# B&R Automation Studio project MotionTestBenchMaster (part 56)

```iecst
                               VAR_DOS_SEQ.Device.LTJ203.ALR_HighLimitEn := FALSE;                                     (* STEP: 115 Hema Tank Level*)
                               VAR_DOS_SEQ.Device.LTJ203.ALR_HighLimitSP := 0;
                               VAR_DOS_SEQ.Device.LTJ203.ALR_LowLimitEn := FALSE;
                               VAR_DOS_SEQ.Device.LTJ203.ALR_LowLimitSP := 0;
                               VAR_DOS_SEQ.Device.LTJ203.SP := 0;
                               VAR_DOS_SEQ.Device.LTJ203.CMP := 0;
                               VAR_DOS_SEQ.Device.LTJ203.MinDev := 0;
                               VAR_DOS_SEQ.Device.LTJ203.MaxDev := 0;

                               VAR_DOS_SEQ.Device.TTJ203.ALR_HighLimitEn := FALSE;                                     (* STEP: 115 Hema Tank Temperature*)
                               VAR_DOS_SEQ.Device.TTJ203.ALR_HighLimitSP := 0;
                               VAR_DOS_SEQ.Device.TTJ203.ALR_LowLimitEn := FALSE;
                               VAR_DOS_SEQ.Device.TTJ203.ALR_LowLimitSP := 0;
                               VAR_DOS_SEQ.Device.TTJ203.SP := 0;
                               VAR_DOS_SEQ.Device.TTJ203.CMP := 0;
                               VAR_DOS_SEQ.Device.TTJ203.MinDev := 0;
                               VAR_DOS_SEQ.Device.TTJ203.MaxDev := 0;

                               VAR_DOS_SEQ.Device.LSJ200.ALR := FALSE;                                                 (* STEP: 115 *)
                               VAR_DOS_SEQ.Device.LSJ200.WAIT_OFF := FALSE;
                               VAR_DOS_SEQ.Device.LSJ200.WAIT_ON := FALSE;

                               VAR_DOS_SEQ.Device.LSJ201.ALR := FALSE;                                                 (* STEP: 115 *)
                               VAR_DOS_SEQ.Device.LSJ201.WAIT_OFF := FALSE;
                               VAR_DOS_SEQ.Device.LSJ201.WAIT_ON := FALSE;

                               VAR_DOS_SEQ.Device.LSJ202.ALR := FALSE;                                                 (* STEP: 115 *)
                               VAR_DOS_SEQ.Device.LSJ202.WAIT_OFF := FALSE;
                               VAR_DOS_SEQ.Device.LSJ202.WAIT_ON := FALSE;

                               VAR_DOS_SEQ.Device.FSJ201.ALR := FALSE;                                                 (* STEP: 115 *)
                               VAR_DOS_SEQ.Device.FSJ201.WAIT_OFF := FALSE;
                               VAR_DOS_SEQ.Device.FSJ201.WAIT_ON := FALSE;

                               VAR_DOS_SEQ.Device.FSJ202.ALR := FALSE;                                                 (* STEP: 115 *)
                               VAR_DOS_SEQ.Device.FSJ202.WAIT_OFF := FALSE;
                               VAR_DOS_SEQ.Device.FSJ202.WAIT_ON := FALSE;

                               VAR_DOS_SEQ.Mem.PBAbortEnable := TRUE;                                                  (* STEP: 115 PB Abort Sequence Enable*)
                               VAR_DOS_SEQ.Mem.PBStopEnable := FALSE;                                                  (* STEP: 115 PB Stop Sequence Enable*)
                               VAR_DOS_SEQ.Mem.PBStartEnable := FALSE;                                                 (* STEP: 115 PB Start Sequence Enable*)
                               VAR_DOS_SEQ.Mem.ContainersStop := TRUE;                                                 (* STEP: 115 *)
                               VAR_DOS_SEQ.Mem.MachineStart := FALSE;                                                  (* STEP: 115 *)
                               VAR_DOS_SEQ.Mem.MachineStop := TRUE;                                                    (* STEP: 115 *)
                               VAR_DOS_SEQ.Mem.DummyBottles := FALSE;                                                  (* STEP: 115 Dummy Bottle Install*)
                               VAR_DOS_SEQ.Mem.PositioningRequest := FALSE;                                            (* STEP: 115 Request of Cam Positioning at height SP of Sequncer*)
                               VAR_DOS_SEQ.Mem.COP_Cycle := FALSE;                                                     (* STEP: 115 COP Cycle Check Requested*)
                               VAR_DOS_SEQ.Mem.LapsCounter := FALSE;                                                   (* STEP: 115 *)
                               VAR_DOS_SEQ.Mem.ValveOpening := FALSE;                                                  (* STEP: 115 *)
                               VAR_DOS_SEQ.Mem.CopAfterCipRequest := FALSE;                                            (* STEP: 115 Request Of Cop After Cip*)

                               VAR_DOS_SEQ.ITC.CIP_CleaningRequest := FALSE;                                           (* STEP: 115 To CIP -> Request of Solution Sending*)
                               VAR_DOS_SEQ.ITC.CIP_Alarm := FALSE;                                                     (* STEP: 115 To CIP -> Critical Alarm Present*)
                               VAR_DOS_SEQ.ITC.CIP_RinseEnded := FALSE;                                                (* STEP: 115 To CIP -> Rinse Finished*)
                               VAR_DOS_SEQ.ITC.CIP_ChangeEnded := FALSE;                                               (* STEP: 115 To CIP -> Change Finished*)
                               VAR_DOS_SEQ.ITC.CIP_DrainRunning := FALSE;                                              (* STEP: 115 To CIP -> Drain Cycle Running*)
                               VAR_DOS_SEQ.ITC.CIP_RinseRunning := FALSE;                                              (* STEP: 115 To CIP -> Rinse Cycle Running*)
                               VAR_DOS_SEQ.ITC.CIP_CleaningRunning := FALSE;                                           (* STEP: 115 To CIP -> Cleaning Cycle Running*)
                               VAR_DOS_SEQ.ITC.CIP_DrainEnded := FALSE;                                                (* STEP: 115 To CIP -> Drain Finished*)
                               VAR_DOS_SEQ.ITC.CIP_FloodingEnded := FALSE;                                             (* STEP: 115 To CIP -> Flooding Finished*)
                               VAR_DOS_SEQ.ITC.CIP_FlipEnable := FALSE;                                                (* STEP: 115 *)
                               VAR_DOS_SEQ.ITC.CIP_CycleEnded := FALSE;                                                (* STEP: 115 *)

                               VAR_DOS_SEQ.ITC.PROD_ReadyForHeating := FALSE;                                          (* STEP: 115 To PASTO -> Filler Ready for Production (Heating)*)
                               VAR_DOS_SEQ.ITC.PROD_DoserInTemperature := FALSE;                                       (* STEP: 115 To PASTO -> Filler Temperature OK (After Heating)*)
                               VAR_DOS_SEQ.ITC.PROD_ProductRequest := FALSE;                                           (* STEP: 115 To PASTO -> Product Request*)
                               VAR_DOS_SEQ.ITC.PROD_DoserOnFillingMode := FALSE;                                       (* STEP: 115 To PASTO -> Product Consumend -Filling Valve Opening*)
                               VAR_DOS_SEQ.ITC.PROD_EndProductionCompleted := FALSE;                                   (* STEP: 115 To PASTO -> End Production Done*)
                               VAR_DOS_SEQ.ITC.PROD_ProductRecoveryEnd := FALSE;                                       (* STEP: 115 To PASTO -> Product Recovery End*)
                               VAR_DOS_SEQ.ITC.PROD_WaterRequestAfterProd := FALSE;                                    (* STEP: 115 To PASTO -> Water Request For Filler Rinse Afetr Production*)

                       116..129: (* Spare Steps *)

                       130: (* DRAIN - Final Drain *)

                               VAR_DOS_SEQ.Device.PPJ201_PID.PID_Enable := FALSE;                                      (* STEP: 130 Doser Recovery Pump*)
                               VAR_DOS_SEQ.Device.PPJ201_PID.PID_Mode := FALSE;
                               VAR_DOS_SEQ.Device.PPJ201_PID.Auto_SP_Value := 0;
                               VAR_DOS_SEQ.Device.PPJ201_PID.FIX_Value := 0;

                               VAR_DOS_SEQ.Device.PPJ202_PID.PID_Enable := FALSE;                                      (* STEP: 130 Doser Recovery Pump*)
                               VAR_DOS_SEQ.Device.PPJ202_PID.PID_Mode := FALSE;
                               VAR_DOS_SEQ.Device.PPJ202_PID.Auto_SP_Value := 0;
                               VAR_DOS_SEQ.Device.PPJ202_PID.FIX_Value := 0;

                               VAR_DOS_SEQ.Device.PPJ203_PID.PID_Enable := FALSE;                                      (* STEP: 130 Diaphragm Pump for Recovery pulp*)
                               VAR_DOS_SEQ.Device.PPJ203_PID.PID_Mode := FALSE;
                               VAR_DOS_SEQ.Device.PPJ203_PID.Auto_SP_Value := 0;
                               VAR_DOS_SEQ.Device.PPJ203_PID.FIX_Value := 0;

                               VAR_DOS_SEQ.Device.MMJ201_PID.PID_Enable := FALSE;                                      (* STEP: 130 Shaker Motor*)
                               VAR_DOS_SEQ.Device.MMJ201_PID.PID_Mode := FALSE;
                               VAR_DOS_SEQ.Device.MMJ201_PID.Auto_SP_Value := 0;
                               VAR_DOS_SEQ.Device.MMJ201_PID.FIX_Value := 0;

                               VAR_DOS_SEQ.Device.RVJ201_PID.PID_Enable := FALSE;                                      (* STEP: 130 *)
                               VAR_DOS_SEQ.Device.RVJ201_PID.PID_Mode := FALSE;
                               VAR_DOS_SEQ.Device.RVJ201_PID.Auto_SP_Value := 0;
                               VAR_DOS_SEQ.Device.RVJ201_PID.FIX_Value := 0;

                               VAR_DOS_SEQ.Device.AVJ201.AutoCnd := FALSE;                                             (* STEP: 130 Inlet Valve*)
                               VAR_DOS_SEQ.Device.AVJ201.EnableCnd := FALSE;
                               VAR_DOS_SEQ.Device.AVJ210.AutoCnd := FALSE;                                             (* STEP: 130 Washing Duct Valve*)
                               VAR_DOS_SEQ.Device.AVJ210.EnableCnd := FALSE;
                               VAR_DOS_SEQ.Device.AVJ211.AutoCnd := FALSE;                                             (* STEP: 130 Sprayball Valve*)
                               VAR_DOS_SEQ.Device.AVJ211.EnableCnd := FALSE;
                               VAR_DOS_SEQ.Device.AVJ212.AutoCnd := FALSE;                                             (* STEP: 130 *)
                               VAR_DOS_SEQ.Device.AVJ212.EnableCnd := FALSE;
                               VAR_DOS_SEQ.Device.AVJ215.AutoCnd := TRUE;                                              (* STEP: 130 Atmospheric drain valve*)
                               VAR_DOS_SEQ.Device.AVJ215.EnableCnd := FALSE;
                               VAR_DOS_SEQ.Device.AVJ216.AutoCnd := FALSE;                                             (* STEP: 130 Recirculation Valve*)
                               VAR_DOS_SEQ.Device.AVJ216.EnableCnd := FALSE;
                               VAR_DOS_SEQ.Device.AVJ217.AutoCnd := TRUE;                                              (* STEP: 130 Tank Hema Drain Valve*)
                               VAR_DOS_SEQ.Device.AVJ217.EnableCnd := FALSE;
                               VAR_DOS_SEQ.Device.AVJ218.AutoCnd := FALSE;                                             (* STEP: 130 Recirculation Valve*)
                               VAR_DOS_SEQ.Device.AVJ218.EnableCnd := FALSE;
                               VAR_DOS_SEQ.Device.AVJ221.AutoCnd := TRUE;                                              (* STEP: 130 Inlet Loop Valve*)
                               VAR_DOS_SEQ.Device.AVJ221.EnableCnd := FALSE;
                               VAR_DOS_SEQ.Device.AVJ230.AutoCnd := FALSE;                                             (* STEP: 130 *)
                               VAR_DOS_SEQ.Device.AVJ230.EnableCnd := FALSE;
                               VAR_DOS_SEQ.Device.AVJ231.AutoCnd := FALSE;                                             (* STEP: 130 *)
                               VAR_DOS_SEQ.Device.AVJ231.EnableCnd := FALSE;
                               VAR_DOS_SEQ.Device.AVJ232.AutoCnd := TRUE;                                              (* STEP: 130 *)
                               VAR_DOS_SEQ.Device.AVJ232.EnableCnd := FALSE;
                               VAR_DOS_SEQ.Device.AVJ233.AutoCnd := FALSE;                                             (* STEP: 130 *)
                               VAR_DOS_SEQ.Device.AVJ233.EnableCnd := FALSE;
                               VAR_DOS_SEQ.Device.AVJ234.AutoCnd := FALSE;                                             (* STEP: 130 *)
                               VAR_DOS_SEQ.Device.AVJ234.EnableCnd := FALSE;
                               VAR_DOS_SEQ.Device.AVJ235.AutoCnd := FALSE;                                             (* STEP: 130 *)
                               VAR_DOS_SEQ.Device.AVJ235.EnableCnd := FALSE;

                               VAR_DOS_SEQ.Device.LTJ203.ALR_HighLimitEn := FALSE;                                     (* STEP: 130 Hema Tank Level*)
                               VAR_DOS_SEQ.Device.LTJ203.ALR_HighLimitSP := 0;
                               VAR_DOS_SEQ.Device.LTJ203.ALR_LowLimitEn := FALSE;
                               VAR_DOS_SEQ.Device.LTJ203.ALR_LowLimitSP := 0;
                               VAR_DOS_SEQ.Device.LTJ203.SP := 0;
                               VAR_DOS_SEQ.Device.LTJ203.CMP := 0;
                               VAR_DOS_SEQ.Device.LTJ203.MinDev := 0;
                               VAR_DOS_SEQ.Device.LTJ203.MaxDev := 0;

                               VAR_DOS_SEQ.Device.TTJ203.ALR_HighLimitEn := FALSE;                                     (* STEP: 130 Hema Tank Temperature*)
                               VAR_DOS_SEQ.Device.TTJ203.ALR_HighLimitSP := 0;
                               VAR_DOS_SEQ.Device.TTJ203.ALR_LowLimitEn := FALSE;
                               VAR_DOS_SEQ.Device.TTJ203.ALR_LowLimitSP := 0;
                               VAR_DOS_SEQ.Device.TTJ203.SP := 0;
                               VAR_DOS_SEQ.Device.TTJ203.CMP := 0;
                               VAR_DOS_SEQ.Device.TTJ203.MinDev := 0;
                               VAR_DOS_SEQ.Device.TTJ203.MaxDev := 0;

                               VAR_DOS_SEQ.Device.LSJ200.ALR := FALSE;                                                 (* STEP: 130 *)
                               VAR_DOS_SEQ.Device.LSJ200.WAIT_OFF := FALSE;
                               VAR_DOS_SEQ.Device.LSJ200.WAIT_ON := FALSE;

                               VAR_DOS_SEQ.Device.LSJ201.ALR := FALSE;                                                 (* STEP: 130 *)
                               VAR_DOS_SEQ.Device.LSJ201.WAIT_OFF := FALSE;
                               VAR_DOS_SEQ.Device.LSJ201.WAIT_ON := FALSE;

                               VAR_DOS_SEQ.Device.LSJ202.ALR := FALSE;                                                 (* STEP: 130 *)
                               VAR_DOS_SEQ.Device.LSJ202.WAIT_OFF := FALSE;
                               VAR_DOS_SEQ.Device.LSJ202.WAIT_ON := FALSE;

                               VAR_DOS_SEQ.Device.FSJ201.ALR := FALSE;                                                 (* STEP: 130 *)
                               VAR_DOS_SEQ.Device.FSJ201.WAIT_OFF := FALSE;
                               VAR_DOS_SEQ.Device.FSJ201.WAIT_ON := FALSE;

                               VAR_DOS_SEQ.Device.FSJ202.ALR := FALSE;                                                 (* STEP: 130 *)
                               VAR_DOS_SEQ.Device.FSJ202.WAIT_OFF := FALSE;
                               VAR_DOS_SEQ.Device.FSJ202.WAIT_ON := FALSE;

                               VAR_DOS_SEQ.Mem.PBAbortEnable := TRUE;                                                  (* STEP: 130 PB Abort Sequence Enable*)
                               VAR_DOS_SEQ.Mem.PBStopEnable := TRUE;                                                   (* STEP: 130 PB Stop Sequence Enable*)
                               VAR_DOS_SEQ.Mem.PBStartEnable := FALSE;                                                 (* STEP: 130 PB Start Sequence Enable*)
                               VAR_DOS_SEQ.Mem.ContainersStop := TRUE;                                                 (* STEP: 130 *)
                               VAR_DOS_SEQ.Mem.MachineStart := TRUE;                                                   (* STEP: 130 *)
                               VAR_DOS_SEQ.Mem.MachineStop := FALSE;                                                   (* STEP: 130 *)
                               VAR_DOS_SEQ.Mem.DummyBottles := FALSE;                                                  (* STEP: 130 Dummy Bottle Install*)
                               VAR_DOS_SEQ.Mem.PositioningRequest := FALSE;                                            (* STEP: 130 Request of Cam Positioning at height SP of Sequncer*)
                               VAR_DOS_SEQ.Mem.COP_Cycle := FALSE;                                                     (* STEP: 130 COP Cycle Check Requested*)
                               VAR_DOS_SEQ.Mem.LapsCounter := FALSE;                                                   (* STEP: 130 *)
                               VAR_DOS_SEQ.Mem.ValveOpening := TRUE;                                                   (* STEP: 130 *)
                               VAR_DOS_SEQ.Mem.CopAfterCipRequest := FALSE;                                            (* STEP: 130 Request Of Cop After Cip*)

                               VAR_DOS_SEQ.ITC.CIP_CleaningRequest := FALSE;                                           (* STEP: 130 To CIP -> Request of Solution Sending*)
                               VAR_DOS_SEQ.ITC.CIP_Alarm := FALSE;                                                     (* STEP: 130 To CIP -> Critical Alarm Present*)
                               VAR_DOS_SEQ.ITC.CIP_RinseEnded := FALSE;                                                (* STEP: 130 To CIP -> Rinse Finished*)
                               VAR_DOS_SEQ.ITC.CIP_ChangeEnded := FALSE;                                               (* STEP: 130 To CIP -> Change Finished*)
                               VAR_DOS_SEQ.ITC.CIP_DrainRunning := FALSE;                                              (* STEP: 130 To CIP -> Drain Cycle Running*)
                               VAR_DOS_SEQ.ITC.CIP_RinseRunning := FALSE;                                              (* STEP: 130 To CIP -> Rinse Cycle Running*)
                               VAR_DOS_SEQ.ITC.CIP_CleaningRunning := FALSE;                                           (* STEP: 130 To CIP -> Cleaning Cycle Running*)
                               VAR_DOS_SEQ.ITC.CIP_DrainEnded := FALSE;                                                (* STEP: 130 To CIP -> Drain Finished*)
                               VAR_DOS_SEQ.ITC.CIP_FloodingEnded := FALSE;                                             (* STEP: 130 To CIP -> Flooding Finished*)
                               VAR_DOS_SEQ.ITC.CIP_FlipEnable := FALSE;                                                (* STEP: 130 *)
                               VAR_DOS_SEQ.ITC.CIP_CycleEnded := FALSE;                                                (* STEP: 130 *)

                               VAR_DOS_SEQ.ITC.PROD_ReadyForHeating := FALSE;                                          (* STEP: 130 To PASTO -> Filler Ready for Production (Heating)*)
                               VAR_DOS_SEQ.ITC.PROD_DoserInTemperature := FALSE;                                       (* STEP: 130 To PASTO -> Filler Temperature OK (After Heating)*)
                               VAR_DOS_SEQ.ITC.PROD_ProductRequest := FALSE;                                           (* STEP: 130 To PASTO -> Product Request*)
                               VAR_DOS_SEQ.ITC.PROD_DoserOnFillingMode := FALSE;                                       (* STEP: 130 To PASTO -> Product Consumend -Filling Valve Opening*)
                               VAR_DOS_SEQ.ITC.PROD_EndProductionCompleted := FALSE;                                   (* STEP: 130 To PASTO -> End Production Done*)
                               VAR_DOS_SEQ.ITC.PROD_ProductRecoveryEnd := FALSE;                                       (* STEP: 130 To PASTO -> Product Recovery End*)
                               VAR_DOS_SEQ.ITC.PROD_WaterRequestAfterProd := FALSE;                                    (* STEP: 130 To PASTO -> Water Request For Filler Rinse Afetr Production*)

                       131: (* DRAIN - Filling valve closing *)

                               VAR_DOS_SEQ.Device.PPJ201_PID.PID_Enable := FALSE;                                      (* STEP: 131 Doser Recovery Pump*)
                               VAR_DOS_SEQ.Device.PPJ201_PID.PID_Mode := FALSE;
                               VAR_DOS_SEQ.Device.PPJ201_PID.Auto_SP_Value := 0;
                               VAR_DOS_SEQ.Device.PPJ201_PID.FIX_Value := 0;

                               VAR_DOS_SEQ.Device.PPJ202_PID.PID_Enable := FALSE;                                      (* STEP: 131 Doser Recovery Pump*)
                               VAR_DOS_SEQ.Device.PPJ202_PID.PID_Mode := FALSE;
                               VAR_DOS_SEQ.Device.PPJ202_PID.Auto_SP_Value := 0;
                               VAR_DOS_SEQ.Device.PPJ202_PID.FIX_Value := 0;

                               VAR_DOS_SEQ.Device.PPJ203_PID.PID_Enable := FALSE;                                      (* STEP: 131 Diaphragm Pump for Recovery pulp*)
                               VAR_DOS_SEQ.Device.PPJ203_PID.PID_Mode := FALSE;
                               VAR_DOS_SEQ.Device.PPJ203_PID.Auto_SP_Value := 0;
                               VAR_DOS_SEQ.Device.PPJ203_PID.FIX_Value := 0;

                               VAR_DOS_SEQ.Device.MMJ201_PID.PID_Enable := FALSE;                                      (* STEP: 131 Shaker Motor*)
                               VAR_DOS_SEQ.Device.MMJ201_PID.PID_Mode := FALSE;
                               VAR_DOS_SEQ.Device.MMJ201_PID.Auto_SP_Value := 0;
                               VAR_DOS_SEQ.Device.MMJ201_PID.FIX_Value := 0;

                               VAR_DOS_SEQ.Device.RVJ201_PID.PID_Enable := FALSE;                                      (* STEP: 131 *)
                               VAR_DOS_SEQ.Device.RVJ201_PID.PID_Mode := FALSE;
                               VAR_DOS_SEQ.Device.RVJ201_PID.Auto_SP_Value := 0;
                               VAR_DOS_SEQ.Device.RVJ201_PID.FIX_Value := 0;

                               VAR_DOS_SEQ.Device.AVJ201.AutoCnd := FALSE;                                             (* STEP: 131 Inlet Valve*)
                               VAR_DOS_SEQ.Device.AVJ201.EnableCnd := FALSE;
                               VAR_DOS_SEQ.Device.AVJ210.AutoCnd := FALSE;                                             (* STEP: 131 Washing Duct Valve*)
                               VAR_DOS_SEQ.Device.AVJ210.EnableCnd := FALSE;
                               VAR_DOS_SEQ.Device.AVJ211.AutoCnd := FALSE;                                             (* STEP: 131 Sprayball Valve*)
                               VAR_DOS_SEQ.Device.AVJ211.EnableCnd := FALSE;
                               VAR_DOS_SEQ.Device.AVJ212.AutoCnd := FALSE;                                             (* STEP: 131 *)
                               VAR_DOS_SEQ.Device.AVJ212.EnableCnd := FALSE;
                               VAR_DOS_SEQ.Device.AVJ215.AutoCnd := TRUE;                                              (* STEP: 131 Atmospheric drain valve*)
                               VAR_DOS_SEQ.Device.AVJ215.EnableCnd := FALSE;
                               VAR_DOS_SEQ.Device.AVJ216.AutoCnd := FALSE;                                             (* STEP: 131 Recirculation Valve*)
                               VAR_DOS_SEQ.Device.AVJ216.EnableCnd := FALSE;
                               VAR_DOS_SEQ.Device.AVJ217.AutoCnd := TRUE;                                              (* STEP: 131 Tank Hema Drain Valve*)
                               VAR_DOS_SEQ.Device.AVJ217.EnableCnd := FALSE;
                               VAR_DOS_SEQ.Device.AVJ218.AutoCnd := FALSE;                                             (* STEP: 131 Recirculation Valve*)
                               VAR_DOS_SEQ.Device.AVJ218.EnableCnd := FALSE;
                               VAR_DOS_SEQ.Device.AVJ221.AutoCnd := FALSE;                                             (* STEP: 131 Inlet Loop Valve*)
                               VAR_DOS_SEQ.Device.AVJ221.EnableCnd := FALSE;
                               VAR_DOS_SEQ.Device.AVJ230.AutoCnd := FALSE;                                             (* STEP: 131 *)
                               VAR_DOS_SEQ.Device.AVJ230.EnableCnd := FALSE;
                               VAR_DOS_SEQ.Device.AVJ231.AutoCnd := FALSE;                                             (* STEP: 131 *)
                               VAR_DOS_SEQ.Device.AVJ231.EnableCnd := FALSE;
                               VAR_DOS_SEQ.Device.AVJ232.AutoCnd := TRUE;                                              (* STEP: 131 *)
                               VAR_DOS_SEQ.Device.AVJ232.EnableCnd := FALSE;
                               VAR_DOS_SEQ.Device.AVJ233.AutoCnd := FALSE;                                             (* STEP: 131 *)
                               VAR_DOS_SEQ.Device.AVJ233.EnableCnd := FALSE;
                               VAR_DOS_SEQ.Device.AVJ234.AutoCnd := FALSE;                                             (* STEP: 131 *)
                               VAR_DOS_SEQ.Device.AVJ234.EnableCnd := FALSE;
                               VAR_DOS_SEQ.Device.AVJ235.AutoCnd := FALSE;                                             (* STEP: 131 *)
                               VAR_DOS_SEQ.Device.AVJ235.EnableCnd := FALSE;

                               VAR_DOS_SEQ.Device.LTJ203.ALR_HighLimitEn := FALSE;                                     (* STEP: 131 Hema Tank Level*)
                               VAR_DOS_SEQ.Device.LTJ203.ALR_HighLimitSP := 0;
                               VAR_DOS_SEQ.Device.LTJ203.ALR_LowLimitEn := FALSE;
                               VAR_DOS_SEQ.Device.LTJ203.ALR_LowLimitSP := 0;
                               VAR_DOS_SEQ.Device.LTJ203.SP := 0;
                               VAR_DOS_SEQ.Device.LTJ203.CMP := 0;
                               VAR_DOS_SEQ.Device.LTJ203.MinDev := 0;
                               VAR_DOS_SEQ.Device.LTJ203.MaxDev := 0;

                               VAR_DOS_SEQ.Device.TTJ203.ALR_HighLimitEn := FALSE;                                     (* STEP: 131 Hema Tank Temperature*)
                               VAR_DOS_SEQ.Device.TTJ203.ALR_HighLimitSP := 0;
                               VAR_DOS_SEQ.Device.TTJ203.ALR_LowLimitEn := FALSE;
                               VAR_DOS_SEQ.Device.TTJ203.ALR_LowLimitSP := 0;
                               VAR_DOS_SEQ.Device.TTJ203.SP := 0;
                               VAR_DOS_SEQ.Device.TTJ203.CMP := 0;
                               VAR_DOS_SEQ.Device.TTJ203.MinDev := 0;
                               VAR_DOS_SEQ.Device.TTJ203.MaxDev := 0;

                               VAR_DOS_SEQ.Device.LSJ200.ALR := FALSE;                                                 (* STEP: 131 *)
                               VAR_DOS_SEQ.Device.LSJ200.WAIT_OFF := FALSE;
                               VAR_DOS_SEQ.Device.LSJ200.WAIT_ON := FALSE;

                               VAR_DOS_SEQ.Device.LSJ201.ALR := FALSE;                                                 (* STEP: 131 *)
                               VAR_DOS_SEQ.Device.LSJ201.WAIT_OFF := FALSE;
                               VAR_DOS_SEQ.Device.LSJ201.WAIT_ON := FALSE;

                               VAR_DOS_SEQ.Device.LSJ202.ALR := FALSE;                                                 (* STEP: 131 *)
                               VAR_DOS_SEQ.Device.LSJ202.WAIT_OFF := FALSE;
                               VAR_DOS_SEQ.Device.LSJ202.WAIT_ON := FALSE;

                               VAR_DOS_SEQ.Device.FSJ201.ALR := FALSE;                                                 (* STEP: 131 *)
                               VAR_DOS_SEQ.Device.FSJ201.WAIT_OFF := FALSE;
                               VAR_DOS_SEQ.Device.FSJ201.WAIT_ON := FALSE;

                               VAR_DOS_SEQ.Device.FSJ202.ALR := FALSE;                                                 (* STEP: 131 *)
                               VAR_DOS_SEQ.Device.FSJ202.WAIT_OFF := FALSE;
                               VAR_DOS_SEQ.Device.FSJ202.WAIT_ON := FALSE;

                               VAR_DOS_SEQ.Mem.PBAbortEnable := TRUE;                                                  (* STEP: 131 PB Abort Sequence Enable*)
                               VAR_DOS_SEQ.Mem.PBStopEnable := TRUE;                                                   (* STEP: 131 PB Stop Sequence Enable*)
                               VAR_DOS_SEQ.Mem.PBStartEnable := FALSE;                                                 (* STEP: 131 PB Start Sequence Enable*)
                               VAR_DOS_SEQ.Mem.ContainersStop := TRUE;                                                 (* STEP: 131 *)
                               VAR_DOS_SEQ.Mem.MachineStart := TRUE;                                                   (* STEP: 131 *)
                               VAR_DOS_SEQ.Mem.MachineStop := FALSE;                                                   (* STEP: 131 *)
                               VAR_DOS_SEQ.Mem.DummyBottles := FALSE;                                                  (* STEP: 131 Dummy Bottle Install*)
                               VAR_DOS_SEQ.Mem.PositioningRequest := FALSE;                                            (* STEP: 131 Request of Cam Positioning at height SP of Sequncer*)
                               VAR_DOS_SEQ.Mem.COP_Cycle := FALSE;                                                     (* STEP: 131 COP Cycle Check Requested*)
                               VAR_DOS_SEQ.Mem.LapsCounter := TRUE;                                                    (* STEP: 131 *)
                               VAR_DOS_SEQ.Mem.ValveOpening := FALSE;                                                  (* STEP: 131 *)
                               VAR_DOS_SEQ.Mem.CopAfterCipRequest := FALSE;                                            (* STEP: 131 Request Of Cop After Cip*)

                               VAR_DOS_SEQ.ITC.CIP_CleaningRequest := FALSE;                                           (* STEP: 131 To CIP -> Request of Solution Sending*)
                               VAR_DOS_SEQ.ITC.CIP_Alarm := FALSE;                                                     (* STEP: 131 To CIP -> Critical Alarm Present*)
                               VAR_DOS_SEQ.ITC.CIP_RinseEnded := FALSE;                                                (* STEP: 131 To CIP -> Rinse Finished*)
                               VAR_DOS_SEQ.ITC.CIP_ChangeEnded := FALSE;                                               (* STEP: 131 To CIP -> Change Finished*)
                               VAR_DOS_SEQ.ITC.CIP_DrainRunning := FALSE;                                              (* STEP: 131 To CIP -> Drain Cycle Running*)
                               VAR_DOS_SEQ.ITC.CIP_RinseRunning := FALSE;                                              (* STEP: 131 To CIP -> Rinse Cycle Running*)
                               VAR_DOS_SEQ.ITC.CIP_CleaningRunning := FALSE;                                           (* STEP: 131 To CIP -> Cleaning Cycle Running*)
                               VAR_DOS_SEQ.ITC.CIP_DrainEnded := FALSE;                                                (* STEP: 131 To CIP -> Drain Finished*)
                               VAR_DOS_SEQ.ITC.CIP_FloodingEnded := FALSE;                                             (* STEP: 131 To CIP -> Flooding Finished*)
                               VAR_DOS_SEQ.ITC.CIP_FlipEnable := FALSE;                                                (* STEP: 131 *)
                               VAR_DOS_SEQ.ITC.CIP_CycleEnded := FALSE;                                                (* STEP: 131 *)

                               VAR_DOS_SEQ.ITC.PROD_ReadyForHeating := FALSE;                                          (* STEP: 131 To PASTO -> Filler Ready for Production (Heating)*)
                               VAR_DOS_SEQ.ITC.PROD_DoserInTemperature := FALSE;                                       (* STEP: 131 To PASTO -> Filler Temperature OK (After Heating)*)
                               VAR_DOS_SEQ.ITC.PROD_ProductRequest := FALSE;                                           (* STEP: 131 To PASTO -> Product Request*)
                               VAR_DOS_SEQ.ITC.PROD_DoserOnFillingMode := FALSE;                                       (* STEP: 131 To PASTO -> Product Consumend -Filling Valve Opening*)
                               VAR_DOS_SEQ.ITC.PROD_EndProductionCompleted := FALSE;                                   (* STEP: 131 To PASTO -> End Production Done*)
                               VAR_DOS_SEQ.ITC.PROD_ProductRecoveryEnd := FALSE;                                       (* STEP: 131 To PASTO -> Product Recovery End*)
                               VAR_DOS_SEQ.ITC.PROD_WaterRequestAfterProd := FALSE;                                    (* STEP: 131 To PASTO -> Water Request For Filler Rinse Afetr Production*)

                       132..134: (* Spare Steps *)

                       135: (* Drain - Stopped *)

                               VAR_DOS_SEQ.Device.PPJ201_PID.PID_Enable := FALSE;                                      (* STEP: 135 Doser Recovery Pump*)
                               VAR_DOS_SEQ.Device.PPJ201_PID.PID_Mode := FALSE;
                               VAR_DOS_SEQ.Device.PPJ201_PID.Auto_SP_Value := 0;
                               VAR_DOS_SEQ.Device.PPJ201_PID.FIX_Value := 0;

                               VAR_DOS_SEQ.Device.PPJ202_PID.PID_Enable := FALSE;                                      (* STEP: 135 Doser Recovery Pump*)
                               VAR_DOS_SEQ.Device.PPJ202_PID.PID_Mode := FALSE;
                               VAR_DOS_SEQ.Device.PPJ202_PID.Auto_SP_Value := 0;
                               VAR_DOS_SEQ.Device.PPJ202_PID.FIX_Value := 0;

                               VAR_DOS_SEQ.Device.PPJ203_PID.PID_Enable := FALSE;                                      (* STEP: 135 Diaphragm Pump for Recovery pulp*)
                               VAR_DOS_SEQ.Device.PPJ203_PID.PID_Mode := FALSE;
                               VAR_DOS_SEQ.Device.PPJ203_PID.Auto_SP_Value := 0;
                               VAR_DOS_SEQ.Device.PPJ203_PID.FIX_Value := 0;

                               VAR_DOS_SEQ.Device.MMJ201_PID.PID_Enable := FALSE;                                      (* STEP: 135 Shaker Motor*)
                               VAR_DOS_SEQ.Device.MMJ201_PID.PID_Mode := FALSE;
                               VAR_DOS_SEQ.Device.MMJ201_PID.Auto_SP_Value := 0;
                               VAR_DOS_SEQ.Device.MMJ201_PID.FIX_Value := 0;

                               VAR_DOS_SEQ.Device.RVJ201_PID.PID_Enable := FALSE;                                      (* STEP: 135 *)
                               VAR_DOS_SEQ.Device.RVJ201_PID.PID_Mode := FALSE;
                               VAR_DOS_SEQ.Device.RVJ201_PID.Auto_SP_Value := 0;
                               VAR_DOS_SEQ.Device.RVJ201_PID.FIX_Value := 0;

                               VAR_DOS_SEQ.Device.AVJ201.AutoCnd := FALSE;                                             (* STEP: 135 Inlet Valve*)
                               VAR_DOS_SEQ.Device.AVJ201.EnableCnd := FALSE;
                               VAR_DOS_SEQ.Device.AVJ210.AutoCnd := FALSE;                                             (* STEP: 135 Washing Duct Valve*)
                               VAR_DOS_SEQ.Device.AVJ210.EnableCnd := FALSE;
                               VAR_DOS_SEQ.Device.AVJ211.AutoCnd := FALSE;                                             (* STEP: 135 Sprayball Valve*)
                               VAR_DOS_SEQ.Device.AVJ211.EnableCnd := FALSE;
                               VAR_DOS_SEQ.Device.AVJ212.AutoCnd := FALSE;                                             (* STEP: 135 *)
                               VAR_DOS_SEQ.Device.AVJ212.EnableCnd := FALSE;
                               VAR_DOS_SEQ.Device.AVJ215.AutoCnd := FALSE;                                             (* STEP: 135 Atmospheric drain valve*)
                               VAR_DOS_SEQ.Device.AVJ215.EnableCnd := FALSE;
                               VAR_DOS_SEQ.Device.AVJ216.AutoCnd := FALSE;                                             (* STEP: 135 Recirculation Valve*)
                               VAR_DOS_SEQ.Device.AVJ216.EnableCnd := FALSE;
                               VAR_DOS_SEQ.Device.AVJ217.AutoCnd := FALSE;                                             (* STEP: 135 Tank Hema Drain Valve*)
                               VAR_DOS_SEQ.Device.AVJ217.EnableCnd := FALSE;
                               VAR_DOS_SEQ.Device.AVJ218.AutoCnd := FALSE;                                             (* STEP: 135 Recirculation Valve*)
                               VAR_DOS_SEQ.Device.AVJ218.EnableCnd := FALSE;
                               VAR_DOS_SEQ.Device.AVJ221.AutoCnd := FALSE;                                             (* STEP: 135 Inlet Loop Valve*)
                               VAR_DOS_SEQ.Device.AVJ221.EnableCnd := FALSE;
                               VAR_DOS_SEQ.Device.AVJ230.AutoCnd := FALSE;                                             (* STEP: 135 *)
                               VAR_DOS_SEQ.Device.AVJ230.EnableCnd := FALSE;
                               VAR_DOS_SEQ.Device.AVJ231.AutoCnd := FALSE;                                             (* STEP: 135 *)
                               VAR_DOS_SEQ.Device.AVJ231.EnableCnd := FALSE;
                               VAR_DOS_SEQ.Device.AVJ232.AutoCnd := FALSE;                                             (* STEP: 135 *)
                               VAR_DOS_SEQ.Device.AVJ232.EnableCnd := FALSE;
                               VAR_DOS_SEQ.Device.AVJ233.AutoCnd := FALSE;                                             (* STEP: 135 *)
                               VAR_DOS_SEQ.Device.AVJ233.EnableCnd := FALSE;
                               VAR_DOS_SEQ.Device.AVJ234.AutoCnd := FALSE;                                             (* STEP: 135 *)
                               VAR_DOS_SEQ.Device.AVJ234.EnableCnd := FALSE;
                               VAR_DOS_SEQ.Device.AVJ235.AutoCnd := FALSE;                                             (* STEP: 135 *)
                               VAR_DOS_SEQ.Device.AVJ235.EnableCnd := FALSE;

                               VAR_DOS_SEQ.Device.LTJ203.ALR_HighLimitEn := FALSE;                                     (* STEP: 135 Hema Tank Level*)
                               VAR_DOS_SEQ.Device.LTJ203.ALR_HighLimitSP := 0;
                               VAR_DOS_SEQ.Device.LTJ203.ALR_LowLimitEn := FALSE;
                               VAR_DOS_SEQ.Device.LTJ203.ALR_LowLimitSP := 0;
                               VAR_DOS_SEQ.Device.LTJ203.SP := 0;
                               VAR_DOS_SEQ.Device.LTJ203.CMP := 0;
                               VAR_DOS_SEQ.Device.LTJ203.MinDev := 0;
                               VAR_DOS_SEQ.Device.LTJ203.MaxDev := 0;

                               VAR_DOS_SEQ.Device.TTJ203.ALR_HighLimitEn := FALSE;                                     (* STEP: 135 Hema Tank Temperature*)
                               VAR_DOS_SEQ.Device.TTJ203.ALR_HighLimitSP := 0;
                               VAR_DOS_SEQ.Device.TTJ203.ALR_LowLimitEn := FALSE;
                               VAR_DOS_SEQ.Device.TTJ203.ALR_LowLimitSP := 0;
                               VAR_DOS_SEQ.Device.TTJ203.SP := 0;
                               VAR_DOS_SEQ.Device.TTJ203.CMP := 0;
                               VAR_DOS_SEQ.Device.TTJ203.MinDev := 0;
                               VAR_DOS_SEQ.Device.TTJ203.MaxDev := 0;

                               VAR_DOS_SEQ.Device.LSJ200.ALR := FALSE;                                                 (* STEP: 135 *)
                               VAR_DOS_SEQ.Device.LSJ200.WAIT_OFF := FALSE;
                               VAR_DOS_SEQ.Device.LSJ200.WAIT_ON := FALSE;

                               VAR_DOS_SEQ.Device.LSJ201.ALR := FALSE;                                                 (* STEP: 135 *)
                               VAR_DOS_SEQ.Device.LSJ201.WAIT_OFF := FALSE;
                               VAR_DOS_SEQ.Device.LSJ201.WAIT_ON := FALSE;

                               VAR_DOS_SEQ.Device.LSJ202.ALR := FALSE;                                                 (* STEP: 135 *)
                               VAR_DOS_SEQ.Device.LSJ202.WAIT_OFF := FALSE;
                               VAR_DOS_SEQ.Device.LSJ202.WAIT_ON := FALSE;

                               VAR_DOS_SEQ.Device.FSJ201.ALR := FALSE;                                                 (* STEP: 135 *)
                               VAR_DOS_SEQ.Device.FSJ201.WAIT_OFF := FALSE;
                               VAR_DOS_SEQ.Device.FSJ201.WAIT_ON := FALSE;

                               VAR_DOS_SEQ.Device.FSJ202.ALR := FALSE;                                                 (* STEP: 135 *)
                               VAR_DOS_SEQ.Device.FSJ202.WAIT_OFF := FALSE;
                               VAR_DOS_SEQ.Device.FSJ202.WAIT_ON := FALSE;

                               VAR_DOS_SEQ.Mem.PBAbortEnable := TRUE;                                                  (* STEP: 135 PB Abort Sequence Enable*)
                               VAR_DOS_SEQ.Mem.PBStopEnable := FALSE;                                                  (* STEP: 135 PB Stop Sequence Enable*)
                               VAR_DOS_SEQ.Mem.PBStartEnable := FALSE;                                                 (* STEP: 135 PB Start Sequence Enable*)
                               VAR_DOS_SEQ.Mem.ContainersStop := TRUE;                                                 (* STEP: 135 *)
                               VAR_DOS_SEQ.Mem.MachineStart := FALSE;                                                  (* STEP: 135 *)
                               VAR_DOS_SEQ.Mem.MachineStop := TRUE;                                                    (* STEP: 135 *)
                               VAR_DOS_SEQ.Mem.DummyBottles := FALSE;                                                  (* STEP: 135 Dummy Bottle Install*)
                               VAR_DOS_SEQ.Mem.PositioningRequest := FALSE;                                            (* STEP: 135 Request of Cam Positioning at height SP of Sequncer*)
                               VAR_DOS_SEQ.Mem.COP_Cycle := FALSE;                                                     (* STEP: 135 COP Cycle Check Requested*)
                               VAR_DOS_SEQ.Mem.LapsCounter := FALSE;                                                   (* STEP: 135 *)
                               VAR_DOS_SEQ.Mem.ValveOpening := FALSE;                                                  (* STEP: 135 *)
                               VAR_DOS_SEQ.Mem.CopAfterCipRequest := FALSE;                                            (* STEP: 135 Request Of Cop After Cip*)

                               VAR_DOS_SEQ.ITC.CIP_CleaningRequest := FALSE;                                           (* STEP: 135 To CIP -> Request of Solution Sending*)
                               VAR_DOS_SEQ.ITC.CIP_Alarm := FALSE;                                                     (* STEP: 135 To CIP -> Critical Alarm Present*)
                               VAR_DOS_SEQ.ITC.CIP_RinseEnded := FALSE;                                                (* STEP: 135 To CIP -> Rinse Finished*)
                               VAR_DOS_SEQ.ITC.CIP_ChangeEnded := FALSE;                                               (* STEP: 135 To CIP -> Change Finished*)
                               VAR_DOS_SEQ.ITC.CIP_DrainRunning := FALSE;                                              (* STEP: 135 To CIP -> Drain Cycle Running*)
                               VAR_DOS_SEQ.ITC.CIP_RinseRunning := FALSE;                                              (* STEP: 135 To CIP -> Rinse Cycle Running*)
                               VAR_DOS_SEQ.ITC.CIP_CleaningRunning := FALSE;                                           (* STEP: 135 To CIP -> Cleaning Cycle Running*)
                               VAR_DOS_SEQ.ITC.CIP_DrainEnded := FALSE;                                                (* STEP: 135 To CIP -> Drain Finished*)
                               VAR_DOS_SEQ.ITC.CIP_FloodingEnded := FALSE;                                             (* STEP: 135 To CIP -> Flooding Finished*)
                               VAR_DOS_SEQ.ITC.CIP_FlipEnable := FALSE;                                                (* STEP: 135 *)
                               VAR_DOS_SEQ.ITC.CIP_CycleEnded := FALSE;                                                (* STEP: 135 *)

                               VAR_DOS_SEQ.ITC.PROD_ReadyForHeating := FALSE;                                          (* STEP: 135 To PASTO -> Filler Ready for Production (Heating)*)
                               VAR_DOS_SEQ.ITC.PROD_DoserInTemperature := FALSE;                                       (* STEP: 135 To PASTO -> Filler Temperature OK (After Heating)*)
                               VAR_DOS_SEQ.ITC.PROD_ProductRequest := FALSE;                                           (* STEP: 135 To PASTO -> Product Request*)
                               VAR_DOS_SEQ.ITC.PROD_DoserOnFillingMode := FALSE;                                       (* STEP: 135 To PASTO -> Product Consumend -Filling Valve Opening*)
                               VAR_DOS_SEQ.ITC.PROD_EndProductionCompleted := FALSE;                                   (* STEP: 135 To PASTO -> End Production Done*)
                               VAR_DOS_SEQ.ITC.PROD_ProductRecoveryEnd := FALSE;                                       (* STEP: 135 To PASTO -> Product Recovery End*)
                               VAR_DOS_SEQ.ITC.PROD_WaterRequestAfterProd := FALSE;                                    (* STEP: 135 To PASTO -> Water Request For Filler Rinse Afetr Production*)

                       136..149: (* Spare Steps *)

                       150: (* BYPASS - Check Request *)

                               VAR_DOS_SEQ.Device.PPJ201_PID.PID_Enable := FALSE;                                      (* STEP: 150 Doser Recovery Pump*)
                               VAR_DOS_SEQ.Device.PPJ201_PID.PID_Mode := FALSE;
                               VAR_DOS_SEQ.Device.PPJ201_PID.Auto_SP_Value := 0;
                               VAR_DOS_SEQ.Device.PPJ201_PID.FIX_Value := 0;

                               VAR_DOS_SEQ.Device.PPJ202_PID.PID_Enable := FALSE;                                      (* STEP: 150 Doser Recovery Pump*)
                               VAR_DOS_SEQ.Device.PPJ202_PID.PID_Mode := FALSE;
                               VAR_DOS_SEQ.Device.PPJ202_PID.Auto_SP_Value := 0;
                               VAR_DOS_SEQ.Device.PPJ202_PID.FIX_Value := 0;

                               VAR_DOS_SEQ.Device.PPJ203_PID.PID_Enable := FALSE;                                      (* STEP: 150 Diaphragm Pump for Recovery pulp*)
                               VAR_DOS_SEQ.Device.PPJ203_PID.PID_Mode := FALSE;
                               VAR_DOS_SEQ.Device.PPJ203_PID.Auto_SP_Value := 0;
                               VAR_DOS_SEQ.Device.PPJ203_PID.FIX_Value := 0;

                               VAR_DOS_SEQ.Device.MMJ201_PID.PID_Enable := FALSE;                                      (* STEP: 150 Shaker Motor*)
                               VAR_DOS_SEQ.Device.MMJ201_PID.PID_Mode := FALSE;
                               VAR_DOS_SEQ.Device.MMJ201_PID.Auto_SP_Value := 0;
                               VAR_DOS_SEQ.Device.MMJ201_PID.FIX_Value := 0;

                               VAR_DOS_SEQ.Device.RVJ201_PID.PID_Enable := FALSE;                                      (* STEP: 150 *)
                               VAR_DOS_SEQ.Device.RVJ201_PID.PID_Mode := FALSE;
                               VAR_DOS_SEQ.Device.RVJ201_PID.Auto_SP_Value := 0;
                               VAR_DOS_SEQ.Device.RVJ201_PID.FIX_Value := 0;

                               VAR_DOS_SEQ.Device.AVJ201.AutoCnd := FALSE;                                             (* STEP: 150 Inlet Valve*)
                               VAR_DOS_SEQ.Device.AVJ201.EnableCnd := FALSE;
                               VAR_DOS_SEQ.Device.AVJ210.AutoCnd := FALSE;                                             (* STEP: 150 Washing Duct Valve*)
                               VAR_DOS_SEQ.Device.AVJ210.EnableCnd := FALSE;
                               VAR_DOS_SEQ.Device.AVJ211.AutoCnd := FALSE;                                             (* STEP: 150 Sprayball Valve*)
                               VAR_DOS_SEQ.Device.AVJ211.EnableCnd := FALSE;
                               VAR_DOS_SEQ.Device.AVJ212.AutoCnd := FALSE;                                             (* STEP: 150 *)
                               VAR_DOS_SEQ.Device.AVJ212.EnableCnd := FALSE;
                               VAR_DOS_SEQ.Device.AVJ215.AutoCnd := FALSE;                                             (* STEP: 150 Atmospheric drain valve*)
                               VAR_DOS_SEQ.Device.AVJ215.EnableCnd := FALSE;
                               VAR_DOS_SEQ.Device.AVJ216.AutoCnd := FALSE;                                             (* STEP: 150 Recirculation Valve*)
                               VAR_DOS_SEQ.Device.AVJ216.EnableCnd := FALSE;
                               VAR_DOS_SEQ.Device.AVJ217.AutoCnd := FALSE;                                             (* STEP: 150 Tank Hema Drain Valve*)
                               VAR_DOS_SEQ.Device.AVJ217.EnableCnd := FALSE;
                               VAR_DOS_SEQ.Device.AVJ218.AutoCnd := FALSE;                                             (* STEP: 150 Recirculation Valve*)
                               VAR_DOS_SEQ.Device.AVJ218.EnableCnd := FALSE;
                               VAR_DOS_SEQ.Device.AVJ221.AutoCnd := FALSE;                                             (* STEP: 150 Inlet Loop Valve*)
                               VAR_DOS_SEQ.Device.AVJ221.EnableCnd := FALSE;
                               VAR_DOS_SEQ.Device.AVJ230.AutoCnd := FALSE;                                             (* STEP: 150 *)
                               VAR_DOS_SEQ.Device.AVJ230.EnableCnd := FALSE;
                               VAR_DOS_SEQ.Device.AVJ231.AutoCnd := FALSE;                                             (* STEP: 150 *)
                               VAR_DOS_SEQ.Device.AVJ231.EnableCnd := FALSE;
                               VAR_DOS_SEQ.Device.AVJ232.AutoCnd := FALSE;                                             (* STEP: 150 *)
                               VAR_DOS_SEQ.Device.AVJ232.EnableCnd := FALSE;
                               VAR_DOS_SEQ.Device.AVJ233.AutoCnd := FALSE;                                             (* STEP: 150 *)
                               VAR_DOS_SEQ.Device.AVJ233.EnableCnd := FALSE;
                               VAR_DOS_SEQ.Device.AVJ234.AutoCnd := FALSE;                                             (* STEP: 150 *)
                               VAR_DOS_SEQ.Device.AVJ234.EnableCnd := FALSE;
                               VAR_DOS_SEQ.Device.AVJ235.AutoCnd := FALSE;                                             (* STEP: 150 *)
                               VAR_DOS_SEQ.Device.AVJ235.EnableCnd := FALSE;

                               VAR_DOS_SEQ.Device.LTJ203.ALR_HighLimitEn := FALSE;                                     (* STEP: 150 Hema Tank Level*)
                               VAR_DOS_SEQ.Device.LTJ203.ALR_HighLimitSP := 0;
                               VAR_DOS_SEQ.Device.LTJ203.ALR_LowLimitEn := FALSE;
                               VAR_DOS_SEQ.Device.LTJ203.ALR_LowLimitSP := 0;
                               VAR_DOS_SEQ.Device.LTJ203.SP := 0;
                               VAR_DOS_SEQ.Device.LTJ203.CMP := 0;
                               VAR_DOS_SEQ.Device.LTJ203.MinDev := 0;
                               VAR_DOS_SEQ.Device.LTJ203.MaxDev := 0;

                               VAR_DOS_SEQ.Device.TTJ203.ALR_HighLimitEn := FALSE;                                     (* STEP: 150 Hema Tank Temperature*)
                               VAR_DOS_SEQ.Device.TTJ203.ALR_HighLimitSP := 0;
                               VAR_DOS_SEQ.Device.TTJ203.ALR_LowLimitEn := FALSE;
                               VAR_DOS_SEQ.Device.TTJ203.ALR_LowLimitSP := 0;
                               VAR_DOS_SEQ.Device.TTJ203.SP := 0;
                               VAR_DOS_SEQ.Device.TTJ203.CMP := 0;
                               VAR_DOS_SEQ.Device.TTJ203.MinDev := 0;
                               VAR_DOS_SEQ.Device.TTJ203.MaxDev := 0;

                               VAR_DOS_SEQ.Device.LSJ200.ALR := FALSE;                                                 (* STEP: 150 *)
                               VAR_DOS_SEQ.Device.LSJ200.WAIT_OFF := FALSE;
                               VAR_DOS_SEQ.Device.LSJ200.WAIT_ON := FALSE;

                               VAR_DOS_SEQ.Device.LSJ201.ALR := FALSE;                                                 (* STEP: 150 *)
                               VAR_DOS_SEQ.Device.LSJ201.WAIT_OFF := FALSE;
                               VAR_DOS_SEQ.Device.LSJ201.WAIT_ON := FALSE;

                               VAR_DOS_SEQ.Device.LSJ202.ALR := FALSE;                                                 (* STEP: 150 *)
                               VAR_DOS_SEQ.Device.LSJ202.WAIT_OFF := FALSE;
                               VAR_DOS_SEQ.Device.LSJ202.WAIT_ON := FALSE;

                               VAR_DOS_SEQ.Device.FSJ201.ALR := FALSE;                                                 (* STEP: 150 *)
                               VAR_DOS_SEQ.Device.FSJ201.WAIT_OFF := FALSE;
                               VAR_DOS_SEQ.Device.FSJ201.WAIT_ON := FALSE;

                               VAR_DOS_SEQ.Device.FSJ202.ALR := FALSE;                                                 (* STEP: 150 *)
                               VAR_DOS_SEQ.Device.FSJ202.WAIT_OFF := FALSE;
                               VAR_DOS_SEQ.Device.FSJ202.WAIT_ON := FALSE;

                               VAR_DOS_SEQ.Mem.PBAbortEnable := FALSE;                                                 (* STEP: 150 PB Abort Sequence Enable*)
                               VAR_DOS_SEQ.Mem.PBStopEnable := TRUE;                                                   (* STEP: 150 PB Stop Sequence Enable*)
                               VAR_DOS_SEQ.Mem.PBStartEnable := FALSE;                                                 (* STEP: 150 PB Start Sequence Enable*)
                               VAR_DOS_SEQ.Mem.ContainersStop := FALSE;                                                (* STEP: 150 *)
                               VAR_DOS_SEQ.Mem.MachineStart := FALSE;                                                  (* STEP: 150 *)
                               VAR_DOS_SEQ.Mem.MachineStop := FALSE;                                                   (* STEP: 150 *)
                               VAR_DOS_SEQ.Mem.DummyBottles := FALSE;                                                  (* STEP: 150 Dummy Bottle Install*)
                               VAR_DOS_SEQ.Mem.PositioningRequest := FALSE;                                            (* STEP: 150 Request of Cam Positioning at height SP of Sequncer*)
                               VAR_DOS_SEQ.Mem.COP_Cycle := FALSE;                                                     (* STEP: 150 COP Cycle Check Requested*)
                               VAR_DOS_SEQ.Mem.LapsCounter := FALSE;                                                   (* STEP: 150 *)
                               VAR_DOS_SEQ.Mem.ValveOpening := FALSE;                                                  (* STEP: 150 *)
                               VAR_DOS_SEQ.Mem.CopAfterCipRequest := FALSE;                                            (* STEP: 150 Request Of Cop After Cip*)

                               VAR_DOS_SEQ.ITC.CIP_CleaningRequest := FALSE;                                           (* STEP: 150 To CIP -> Request of Solution Sending*)
                               VAR_DOS_SEQ.ITC.CIP_Alarm := FALSE;                                                     (* STEP: 150 To CIP -> Critical Alarm Present*)
                               VAR_DOS_SEQ.ITC.CIP_RinseEnded := FALSE;                                                (* STEP: 150 To CIP -> Rinse Finished*)
                               VAR_DOS_SEQ.ITC.CIP_ChangeEnded := FALSE;                                               (* STEP: 150 To CIP -> Change Finished*)
                               VAR_DOS_SEQ.ITC.CIP_DrainRunning := FALSE;                                              (* STEP: 150 To CIP -> Drain Cycle Running*)
                               VAR_DOS_SEQ.ITC.CIP_RinseRunning := FALSE;                                              (* STEP: 150 To CIP -> Rinse Cycle Running*)
                               VAR_DOS_SEQ.ITC.CIP_CleaningRunning := FALSE;                                           (* STEP: 150 To CIP -> Cleaning Cycle Running*)
                               VAR_DOS_SEQ.ITC.CIP_DrainEnded := FALSE;                                                (* STEP: 150 To CIP -> Drain Finished*)
                               VAR_DOS_SEQ.ITC.CIP_FloodingEnded := FALSE;                                             (* STEP: 150 To CIP -> Flooding Finished*)
                               VAR_DOS_SEQ.ITC.CIP_FlipEnable := FALSE;                                                (* STEP: 150 *)
                               VAR_DOS_SEQ.ITC.CIP_CycleEnded := FALSE;                                                (* STEP: 150 *)

                               VAR_DOS_SEQ.ITC.PROD_ReadyForHeating := FALSE;                                          (* STEP: 150 To PASTO -> Filler Ready for Production (Heating)*)
                               VAR_DOS_SEQ.ITC.PROD_DoserInTemperature := FALSE;                                       (* STEP: 150 To PASTO -> Filler Temperature OK (After Heating)*)
                               VAR_DOS_SEQ.ITC.PROD_ProductRequest := FALSE;                                           (* STEP: 150 To PASTO -> Product Request*)
                               VAR_DOS_SEQ.ITC.PROD_DoserOnFillingMode := FALSE;                                       (* STEP: 150 To PASTO -> Product Consumend -Filling Valve Opening*)
                               VAR_DOS_SEQ.ITC.PROD_EndProductionCompleted := FALSE;                                   (* STEP: 150 To PASTO -> End Production Done*)
                               VAR_DOS_SEQ.ITC.PROD_ProductRecoveryEnd := FALSE;                                       (* STEP: 150 To PASTO -> Product Recovery End*)
                               VAR_DOS_SEQ.ITC.PROD_WaterRequestAfterProd := FALSE;                                    (* STEP: 150 To PASTO -> Water Request For Filler Rinse Afetr Production*)

                       151: (* BYPASS - Waiting for machine Stop *)

                               VAR_DOS_SEQ.Device.PPJ201_PID.PID_Enable := FALSE;                                      (* STEP: 151 Doser Recovery Pump*)
                               VAR_DOS_SEQ.Device.PPJ201_PID.PID_Mode := FALSE;
                               VAR_DOS_SEQ.Device.PPJ201_PID.Auto_SP_Value := 0;
                               VAR_DOS_SEQ.Device.PPJ201_PID.FIX_Value := 0;

                               VAR_DOS_SEQ.Device.PPJ202_PID.PID_Enable := FALSE;                                      (* STEP: 151 Doser Recovery Pump*)
                               VAR_DOS_SEQ.Device.PPJ202_PID.PID_Mode := FALSE;
                               VAR_DOS_SEQ.Device.PPJ202_PID.Auto_SP_Value := 0;
                               VAR_DOS_SEQ.Device.PPJ202_PID.FIX_Value := 0;

                               VAR_DOS_SEQ.Device.PPJ203_PID.PID_Enable := FALSE;                                      (* STEP: 151 Diaphragm Pump for Recovery pulp*)
                               VAR_DOS_SEQ.Device.PPJ203_PID.PID_Mode := FALSE;
                               VAR_DOS_SEQ.Device.PPJ203_PID.Auto_SP_Value := 0;
                               VAR_DOS_SEQ.Device.PPJ203_PID.FIX_Value := 0;

                               VAR_DOS_SEQ.Device.MMJ201_PID.PID_Enable := FALSE;                                      (* STEP: 151 Shaker Motor*)
                               VAR_DOS_SEQ.Device.MMJ201_PID.PID_Mode := FALSE;
                               VAR_DOS_SEQ.Device.MMJ201_PID.Auto_SP_Value := 0;
                               VAR_DOS_SEQ.Device.MMJ201_PID.FIX_Value := 0;

                               VAR_DOS_SEQ.Device.RVJ201_PID.PID_Enable := FALSE;                                      (* STEP: 151 *)
                               VAR_DOS_SEQ.Device.RVJ201_PID.PID_Mode := FALSE;
                               VAR_DOS_SEQ.Device.RVJ201_PID.Auto_SP_Value := 0;
                               VAR_DOS_SEQ.Device.RVJ201_PID.FIX_Value := 0;

                               VAR_DOS_SEQ.Device.AVJ201.AutoCnd := FALSE;                                             (* STEP: 151 Inlet Valve*)
                               VAR_DOS_SEQ.Device.AVJ201.EnableCnd := FALSE;
                               VAR_DOS_SEQ.Device.AVJ210.AutoCnd := FALSE;                                             (* STEP: 151 Washing Duct Valve*)
                               VAR_DOS_SEQ.Device.AVJ210.EnableCnd := FALSE;
                               VAR_DOS_SEQ.Device.AVJ211.AutoCnd := FALSE;                                             (* STEP: 151 Sprayball Valve*)
                               VAR_DOS_SEQ.Device.AVJ211.EnableCnd := FALSE;
                               VAR_DOS_SEQ.Device.AVJ212.AutoCnd := FALSE;                                             (* STEP: 151 *)
                               VAR_DOS_SEQ.Device.AVJ212.EnableCnd := FALSE;
                               VAR_DOS_SEQ.Device.AVJ215.AutoCnd := FALSE;                                             (* STEP: 151 Atmospheric drain valve*)
                               VAR_DOS_SEQ.Device.AVJ215.EnableCnd := FALSE;
                               VAR_DOS_SEQ.Device.AVJ216.AutoCnd := FALSE;                                             (* STEP: 151 Recirculation Valve*)
                               VAR_DOS_SEQ.Device.AVJ216.EnableCnd := FALSE;
                               VAR_DOS_SEQ.Device.AVJ217.AutoCnd := FALSE;                                             (* STEP: 151 Tank Hema Drain Valve*)
                               VAR_DOS_SEQ.Device.AVJ217.EnableCnd := FALSE;
                               VAR_DOS_SEQ.Device.AVJ218.AutoCnd := FALSE;                                             (* STEP: 151 Recirculation Valve*)
                               VAR_DOS_SEQ.Device.AVJ218.EnableCnd := FALSE;
                               VAR_DOS_SEQ.Device.AVJ221.AutoCnd := FALSE;                                             (* STEP: 151 Inlet Loop Valve*)
                               VAR_DOS_SEQ.Device.AVJ221.EnableCnd := FALSE;
                               VAR_DOS_SEQ.Device.AVJ230.AutoCnd := FALSE;                                             (* STEP: 151 *)
                               VAR_DOS_SEQ.Device.AVJ230.EnableCnd := FALSE;
                               VAR_DOS_SEQ.Device.AVJ231.AutoCnd := FALSE;                                             (* STEP: 151 *)
                               VAR_DOS_SEQ.Device.AVJ231.EnableCnd := FALSE;
                               VAR_DOS_SEQ.Device.AVJ232.AutoCnd := FALSE;                                             (* STEP: 151 *)
                               VAR_DOS_SEQ.Device.AVJ232.EnableCnd := FALSE;
                               VAR_DOS_SEQ.Device.AVJ233.AutoCnd := FALSE;                                             (* STEP: 151 *)
                               VAR_DOS_SEQ.Device.AVJ233.EnableCnd := FALSE;
                               VAR_DOS_SEQ.Device.AVJ234.AutoCnd := FALSE;                                             (* STEP: 151 *)
                               VAR_DOS_SEQ.Device.AVJ234.EnableCnd := FALSE;
                               VAR_DOS_SEQ.Device.AVJ235.AutoCnd := FALSE;                                             (* STEP: 151 *)
                               VAR_DOS_SEQ.Device.AVJ235.EnableCnd := FALSE;

                               VAR_DOS_SEQ.Device.LTJ203.ALR_HighLimitEn := FALSE;                                     (* STEP: 151 Hema Tank Level*)
                               VAR_DOS_SEQ.Device.LTJ203.ALR_HighLimitSP := 0;
                               VAR_DOS_SEQ.Device.LTJ203.ALR_LowLimitEn := FALSE;
                               VAR_DOS_SEQ.Device.LTJ203.ALR_LowLimitSP := 0;
                               VAR_DOS_SEQ.Device.LTJ203.SP := 0;
                               VAR_DOS_SEQ.Device.LTJ203.CMP := 0;
                               VAR_DOS_SEQ.Device.LTJ203.MinDev := 0;
                               VAR_DOS_SEQ.Device.LTJ203.MaxDev := 0;

                               VAR_DOS_SEQ.Device.TTJ203.ALR_HighLimitEn := FALSE;                                     (* STEP: 151 Hema Tank Temperature*)
                               VAR_DOS_SEQ.Device.TTJ203.ALR_HighLimitSP := 0;
                               VAR_DOS_SEQ.Device.TTJ203.ALR_LowLimitEn := FALSE;
                               VAR_DOS_SEQ.Device.TTJ203.ALR_LowLimitSP := 0;
                               VAR_DOS_SEQ.Device.TTJ203.SP := 0;
                               VAR_DOS_SEQ.Device.TTJ203.CMP := 0;
                               VAR_DOS_SEQ.Device.TTJ203.MinDev := 0;
                               VAR_DOS_SEQ.Device.TTJ203.MaxDev := 0;

                               VAR_DOS_SEQ.Device.LSJ200.ALR := FALSE;                                                 (* STEP: 151 *)
                               VAR_DOS_SEQ.Device.LSJ200.WAIT_OFF := FALSE;
                               VAR_DOS_SEQ.Device.LSJ200.WAIT_ON := FALSE;

                               VAR_DOS_SEQ.Device.LSJ201.ALR := FALSE;                                                 (* STEP: 151 *)
                               VAR_DOS_SEQ.Device.LSJ201.WAIT_OFF := FALSE;
                               VAR_DOS_SEQ.Device.LSJ201.WAIT_ON := FALSE;

                               VAR_DOS_SEQ.Device.LSJ202.ALR := FALSE;                                                 (* STEP: 151 *)
                               VAR_DOS_SEQ.Device.LSJ202.WAIT_OFF := FALSE;
                               VAR_DOS_SEQ.Device.LSJ202.WAIT_ON := FALSE;

                               VAR_DOS_SEQ.Device.FSJ201.ALR := FALSE;                                                 (* STEP: 151 *)
                               VAR_DOS_SEQ.Device.FSJ201.WAIT_OFF := FALSE;
                               VAR_DOS_SEQ.Device.FSJ201.WAIT_ON := FALSE;

                               VAR_DOS_SEQ.Device.FSJ202.ALR := FALSE;                                                 (* STEP: 151 *)
                               VAR_DOS_SEQ.Device.FSJ202.WAIT_OFF := FALSE;
                               VAR_DOS_SEQ.Device.FSJ202.WAIT_ON := FALSE;

                               VAR_DOS_SEQ.Mem.PBAbortEnable := FALSE;                                                 (* STEP: 151 PB Abort Sequence Enable*)
                               VAR_DOS_SEQ.Mem.PBStopEnable := TRUE;                                                   (* STEP: 151 PB Stop Sequence Enable*)
                               VAR_DOS_SEQ.Mem.PBStartEnable := FALSE;                                                 (* STEP: 151 PB Start Sequence Enable*)
                               VAR_DOS_SEQ.Mem.ContainersStop := FALSE;                                                (* STEP: 151 *)
                               VAR_DOS_SEQ.Mem.MachineStart := FALSE;                                                  (* STEP: 151 *)
                               VAR_DOS_SEQ.Mem.MachineStop := FALSE;                                                   (* STEP: 151 *)
                               VAR_DOS_SEQ.Mem.DummyBottles := FALSE;                                                  (* STEP: 151 Dummy Bottle Install*)
                               VAR_DOS_SEQ.Mem.PositioningRequest := FALSE;                                            (* STEP: 151 Request of Cam Positioning at height SP of Sequncer*)
                               VAR_DOS_SEQ.Mem.COP_Cycle := FALSE;                                                     (* STEP: 151 COP Cycle Check Requested*)
                               VAR_DOS_SEQ.Mem.LapsCounter := FALSE;                                                   (* STEP: 151 *)
                               VAR_DOS_SEQ.Mem.ValveOpening := FALSE;                                                  (* STEP: 151 *)
                               VAR_DOS_SEQ.Mem.CopAfterCipRequest := FALSE;                                            (* STEP: 151 Request Of Cop After Cip*)

                               VAR_DOS_SEQ.ITC.CIP_CleaningRequest := FALSE;                                           (* STEP: 151 To CIP -> Request of Solution Sending*)
                               VAR_DOS_SEQ.ITC.CIP_Alarm := FALSE;                                                     (* STEP: 151 To CIP -> Critical Alarm Present*)
                               VAR_DOS_SEQ.ITC.CIP_RinseEnded := FALSE;                                                (* STEP: 151 To CIP -> Rinse Finished*)
                               VAR_DOS_SEQ.ITC.CIP_ChangeEnded := FALSE;                                               (* STEP: 151 To CIP -> Change Finished*)
                               VAR_DOS_SEQ.ITC.CIP_DrainRunning := FALSE;                                              (* STEP: 151 To CIP -> Drain Cycle Running*)
                               VAR_DOS_SEQ.ITC.CIP_RinseRunning := FALSE;                                              (* STEP: 151 To CIP -> Rinse Cycle Running*)
                               VAR_DOS_SEQ.ITC.CIP_CleaningRunning := FALSE;                                           (* STEP: 151 To CIP -> Cleaning Cycle Running*)
                               VAR_DOS_SEQ.ITC.CIP_DrainEnded := FALSE;                                                (* STEP: 151 To CIP -> Drain Finished*)
                               VAR_DOS_SEQ.ITC.CIP_FloodingEnded := FALSE;                                             (* STEP: 151 To CIP -> Flooding Finished*)
                               VAR_DOS_SEQ.ITC.CIP_FlipEnable := FALSE;                                                (* STEP: 151 *)
                               VAR_DOS_SEQ.ITC.CIP_CycleEnded := FALSE;                                                (* STEP: 151 *)

                               VAR_DOS_SEQ.ITC.PROD_ReadyForHeating := FALSE;                                          (* STEP: 151 To PASTO -> Filler Ready for Production (Heating)*)
                               VAR_DOS_SEQ.ITC.PROD_DoserInTemperature := FALSE;                                       (* STEP: 151 To PASTO -> Filler Temperature OK (After Heating)*)
                               VAR_DOS_SEQ.ITC.PROD_ProductRequest := FALSE;                                           (* STEP: 151 To PASTO -> Product Request*)
                               VAR_DOS_SEQ.ITC.PROD_DoserOnFillingMode := FALSE;                                       (* STEP: 151 To PASTO -> Product Consumend -Filling Valve Opening*)
                               VAR_DOS_SEQ.ITC.PROD_EndProductionCompleted := FALSE;                                   (* STEP: 151 To PASTO -> End Production Done*)
                               VAR_DOS_SEQ.ITC.PROD_ProductRecoveryEnd := FALSE;                                       (* STEP: 151 To PASTO -> Product Recovery End*)
                               VAR_DOS_SEQ.ITC.PROD_WaterRequestAfterProd := FALSE;                                    (* STEP: 151 To PASTO -> Water Request For Filler Rinse Afetr Production*)

                       152: (* BYPASS - Doser Bypassed *)

                               VAR_DOS_SEQ.Device.PPJ201_PID.PID_Enable := FALSE;                                      (* STEP: 152 Doser Recovery Pump*)
                               VAR_DOS_SEQ.Device.PPJ201_PID.PID_Mode := FALSE;
                               VAR_DOS_SEQ.Device.PPJ201_PID.Auto_SP_Value := 0;
                               VAR_DOS_SEQ.Device.PPJ201_PID.FIX_Value := 0;

                               VAR_DOS_SEQ.Device.PPJ202_PID.PID_Enable := FALSE;                                      (* STEP: 152 Doser Recovery Pump*)
                               VAR_DOS_SEQ.Device.PPJ202_PID.PID_Mode := FALSE;
                               VAR_DOS_SEQ.Device.PPJ202_PID.Auto_SP_Value := 0;
                               VAR_DOS_SEQ.Device.PPJ202_PID.FIX_Value := 0;

                               VAR_DOS_SEQ.Device.PPJ203_PID.PID_Enable := FALSE;                                      (* STEP: 152 Diaphragm Pump for Recovery pulp*)
                               VAR_DOS_SEQ.Device.PPJ203_PID.PID_Mode := FALSE;
                               VAR_DOS_SEQ.Device.PPJ203_PID.Auto_SP_Value := 0;
                               VAR_DOS_SEQ.Device.PPJ203_PID.FIX_Value := 0;

                               VAR_DOS_SEQ.Device.MMJ201_PID.PID_Enable := FALSE;                                      (* STEP: 152 Shaker Motor*)
                               VAR_DOS_SEQ.Device.MMJ201_PID.PID_Mode := FALSE;
                               VAR_DOS_SEQ.Device.MMJ201_PID.Auto_SP_Value := 0;
                               VAR_DOS_SEQ.Device.MMJ201_PID.FIX_Value := 0;

                               VAR_DOS_SEQ.Device.RVJ201_PID.PID_Enable := FALSE;                                      (* STEP: 152 *)
                               VAR_DOS_SEQ.Device.RVJ201_PID.PID_Mode := FALSE;
                               VAR_DOS_SEQ.Device.RVJ201_PID.Auto_SP_Value := 0;
                               VAR_DOS_SEQ.Device.RVJ201_PID.FIX_Value := 0;

                               VAR_DOS_SEQ.Device.AVJ201.AutoCnd := FALSE;                                             (* STEP: 152 Inlet Valve*)
                               VAR_DOS_SEQ.Device.AVJ201.EnableCnd := FALSE;
                               VAR_DOS_SEQ.Device.AVJ210.AutoCnd := FALSE;                                             (* STEP: 152 Washing Duct Valve*)
                               VAR_DOS_SEQ.Device.AVJ210.EnableCnd := FALSE;
                               VAR_DOS_SEQ.Device.AVJ211.AutoCnd := FALSE;                                             (* STEP: 152 Sprayball Valve*)
                               VAR_DOS_SEQ.Device.AVJ211.EnableCnd := FALSE;
                               VAR_DOS_SEQ.Device.AVJ212.AutoCnd := FALSE;                                             (* STEP: 152 *)
                               VAR_DOS_SEQ.Device.AVJ212.EnableCnd := FALSE;
                               VAR_DOS_SEQ.Device.AVJ215.AutoCnd := FALSE;                                             (* STEP: 152 Atmospheric drain valve*)
                               VAR_DOS_SEQ.Device.AVJ215.EnableCnd := FALSE;
                               VAR_DOS_SEQ.Device.AVJ216.AutoCnd := FALSE;                                             (* STEP: 152 Recirculation Valve*)
                               VAR_DOS_SEQ.Device.AVJ216.EnableCnd := FALSE;
                               VAR_DOS_SEQ.Device.AVJ217.AutoCnd := FALSE;                                             (* STEP: 152 Tank Hema Drain Valve*)
                               VAR_DOS_SEQ.Device.AVJ217.EnableCnd := FALSE;
                               VAR_DOS_SEQ.Device.AVJ218.AutoCnd := FALSE;                                             (* STEP: 152 Recirculation Valve*)
                               VAR_DOS_SEQ.Device.AVJ218.EnableCnd := FALSE;
                               VAR_DOS_SEQ.Device.AVJ221.AutoCnd := FALSE;                                             (* STEP: 152 Inlet Loop Valve*)
                               VAR_DOS_SEQ.Device.AVJ221.EnableCnd := FALSE;
                               VAR_DOS_SEQ.Device.AVJ230.AutoCnd := FALSE;                                             (* STEP: 152 *)
                               VAR_DOS_SEQ.Device.AVJ230.EnableCnd := FALSE;
                               VAR_DOS_SEQ.Device.AVJ231.AutoCnd := FALSE;                                             (* STEP: 152 *)
                               VAR_DOS_SEQ.Device.AVJ231.EnableCnd := FALSE;
                               VAR_DOS_SEQ.Device.AVJ232.AutoCnd := FALSE;                                             (* STEP: 152 *)
                               VAR_DOS_SEQ.Device.AVJ232.EnableCnd := FALSE;
                               VAR_DOS_SEQ.Device.AVJ233.AutoCnd := FALSE;                                             (* STEP: 152 *)
                               VAR_DOS_SEQ.Device.AVJ233.EnableCnd := FALSE;
                               VAR_DOS_SEQ.Device.AVJ234.AutoCnd := FALSE;                                             (* STEP: 152 *)
                               VAR_DOS_SEQ.Device.AVJ234.EnableCnd := FALSE;
                               VAR_DOS_SEQ.Device.AVJ235.AutoCnd := FALSE;                                             (* STEP: 152 *)
                               VAR_DOS_SEQ.Device.AVJ235.EnableCnd := FALSE;

                               VAR_DOS_SEQ.Device.LTJ203.ALR_HighLimitEn := FALSE;                                     (* STEP: 152 Hema Tank Level*)
                               VAR_DOS_SEQ.Device.LTJ203.ALR_HighLimitSP := 0;
                               VAR_DOS_SEQ.Device.LTJ203.ALR_LowLimitEn := FALSE;
                               VAR_DOS_SEQ.Device.LTJ203.ALR_LowLimitSP := 0;
                               VAR_DOS_SEQ.Device.LTJ203.SP := 0;
                               VAR_DOS_SEQ.Device.LTJ203.CMP := 0;
                               VAR_DOS_SEQ.Device.LTJ203.MinDev := 0;
                               VAR_DOS_SEQ.Device.LTJ203.MaxDev := 0;

                               VAR_DOS_SEQ.Device.TTJ203.ALR_HighLimitEn := FALSE;                                     (* STEP: 152 Hema Tank Temperature*)
                               VAR_DOS_SEQ.Device.TTJ203.ALR_HighLimitSP := 0;
                               VAR_DOS_SEQ.Device.TTJ203.ALR_LowLimitEn := FALSE;
                               VAR_DOS_SEQ.Device.TTJ203.ALR_LowLimitSP := 0;
                               VAR_DOS_SEQ.Device.TTJ203.SP := 0;
                               VAR_DOS_SEQ.Device.TTJ203.CMP := 0;
                               VAR_DOS_SEQ.Device.TTJ203.MinDev := 0;
                               VAR_DOS_SEQ.Device.TTJ203.MaxDev := 0;

                               VAR_DOS_SEQ.Device.LSJ200.ALR := FALSE;                                                 (* STEP: 152 *)
                               VAR_DOS_SEQ.Device.LSJ200.WAIT_OFF := FALSE;
                               VAR_DOS_SEQ.Device.LSJ200.WAIT_ON := FALSE;

                               VAR_DOS_SEQ.Device.LSJ201.ALR := FALSE;                                                 (* STEP: 152 *)
                               VAR_DOS_SEQ.Device.LSJ201.WAIT_OFF := FALSE;
                               VAR_DOS_SEQ.Device.LSJ201.WAIT_ON := FALSE;

                               VAR_DOS_SEQ.Device.LSJ202.ALR := FALSE;                                                 (* STEP: 152 *)
                               VAR_DOS_SEQ.Device.LSJ202.WAIT_OFF := FALSE;
                               VAR_DOS_SEQ.Device.LSJ202.WAIT_ON := FALSE;

                               VAR_DOS_SEQ.Device.FSJ201.ALR := FALSE;                                                 (* STEP: 152 *)
                               VAR_DOS_SEQ.Device.FSJ201.WAIT_OFF := FALSE;
                               VAR_DOS_SEQ.Device.FSJ201.WAIT_ON := FALSE;

                               VAR_DOS_SEQ.Device.FSJ202.ALR := FALSE;                                                 (* STEP: 152 *)
                               VAR_DOS_SEQ.Device.FSJ202.WAIT_OFF := FALSE;
                               VAR_DOS_SEQ.Device.FSJ202.WAIT_ON := FALSE;

                               VAR_DOS_SEQ.Mem.PBAbortEnable := FALSE;                                                 (* STEP: 152 PB Abort Sequence Enable*)
                               VAR_DOS_SEQ.Mem.PBStopEnable := TRUE;                                                   (* STEP: 152 PB Stop Sequence Enable*)
                               VAR_DOS_SEQ.Mem.PBStartEnable := FALSE;                                                 (* STEP: 152 PB Start Sequence Enable*)
                               VAR_DOS_SEQ.Mem.ContainersStop := FALSE;                                                (* STEP: 152 *)
                               VAR_DOS_SEQ.Mem.MachineStart := FALSE;                                                  (* STEP: 152 *)
                               VAR_DOS_SEQ.Mem.MachineStop := FALSE;                                                   (* STEP: 152 *)
                               VAR_DOS_SEQ.Mem.DummyBottles := FALSE;                                                  (* STEP: 152 Dummy Bottle Install*)
                               VAR_DOS_SEQ.Mem.PositioningRequest := FALSE;                                            (* STEP: 152 Request of Cam Positioning at height SP of Sequncer*)
                               VAR_DOS_SEQ.Mem.COP_Cycle := FALSE;                                                     (* STEP: 152 COP Cycle Check Requested*)
                               VAR_DOS_SEQ.Mem.LapsCounter := FALSE;                                                   (* STEP: 152 *)
                               VAR_DOS_SEQ.Mem.ValveOpening := FALSE;                                                  (* STEP: 152 *)
                               VAR_DOS_SEQ.Mem.CopAfterCipRequest := FALSE;                                            (* STEP: 152 Request Of Cop After Cip*)

                               VAR_DOS_SEQ.ITC.CIP_CleaningRequest := FALSE;                                           (* STEP: 152 To CIP -> Request of Solution Sending*)
                               VAR_DOS_SEQ.ITC.CIP_Alarm := FALSE;                                                     (* STEP: 152 To CIP -> Critical Alarm Present*)
                               VAR_DOS_SEQ.ITC.CIP_RinseEnded := FALSE;                                                (* STEP: 152 To CIP -> Rinse Finished*)
                               VAR_DOS_SEQ.ITC.CIP_ChangeEnded := FALSE;                                               (* STEP: 152 To CIP -> Change Finished*)
                               VAR_DOS_SEQ.ITC.CIP_DrainRunning := FALSE;                                              (* STEP: 152 To CIP -> Drain Cycle Running*)
                               VAR_DOS_SEQ.ITC.CIP_RinseRunning := FALSE;                                              (* STEP: 152 To CIP -> Rinse Cycle Running*)
                               VAR_DOS_SEQ.ITC.CIP_CleaningRunning := FALSE;                                           (* STEP: 152 To CIP -> Cleaning Cycle Running*)
                               VAR_DOS_SEQ.ITC.CIP_DrainEnded := FALSE;                                                (* STEP: 152 To CIP -> Drain Finished*)
                               VAR_DOS_SEQ.ITC.CIP_FloodingEnded := FALSE;                                             (* STEP: 152 To CIP -> Flooding Finished*)
                               VAR_DOS_SEQ.ITC.CIP_FlipEnable := FALSE;                                                (* STEP: 152 *)
                               VAR_DOS_SEQ.ITC.CIP_CycleEnded := FALSE;                                                (* STEP: 152 *)

                               VAR_DOS_SEQ.ITC.PROD_ReadyForHeating := FALSE;                                          (* STEP: 152 To PASTO -> Filler Ready for Production (Heating)*)
                               VAR_DOS_SEQ.ITC.PROD_DoserInTemperature := FALSE;                                       (* STEP: 152 To PASTO -> Filler Temperature OK (After Heating)*)
                               VAR_DOS_SEQ.ITC.PROD_ProductRequest := FALSE;                                           (* STEP: 152 To PASTO -> Product Request*)
                               VAR_DOS_SEQ.ITC.PROD_DoserOnFillingMode := FALSE;                                       (* STEP: 152 To PASTO -> Product Consumend -Filling Valve Opening*)
                               VAR_DOS_SEQ.ITC.PROD_EndProductionCompleted := FALSE;                                   (* STEP: 152 To PASTO -> End Production Done*)
                               VAR_DOS_SEQ.ITC.PROD_ProductRecoveryEnd := FALSE;                                       (* STEP: 152 To PASTO -> Product Recovery End*)
                               VAR_DOS_SEQ.ITC.PROD_WaterRequestAfterProd := FALSE;                                    (* STEP: 152 To PASTO -> Water Request For Filler Rinse Afetr Production*)

                       153: (* BYPASS - Doser Included *)

                               VAR_DOS_SEQ.Device.PPJ201_PID.PID_Enable := FALSE;                                      (* STEP: 153 Doser Recovery Pump*)
                               VAR_DOS_SEQ.Device.PPJ201_PID.PID_Mode := FALSE;
                               VAR_DOS_SEQ.Device.PPJ201_PID.Auto_SP_Value := 0;
                               VAR_DOS_SEQ.Device.PPJ201_PID.FIX_Value := 0;

                               VAR_DOS_SEQ.Device.PPJ202_PID.PID_Enable := FALSE;                                      (* STEP: 153 Doser Recovery Pump*)
                               VAR_DOS_SEQ.Device.PPJ202_PID.PID_Mode := FALSE;
                               VAR_DOS_SEQ.Device.PPJ202_PID.Auto_SP_Value := 0;
                               VAR_DOS_SEQ.Device.PPJ202_PID.FIX_Value := 0;

                               VAR_DOS_SEQ.Device.PPJ203_PID.PID_Enable := FALSE;                                      (* STEP: 153 Diaphragm Pump for Recovery pulp*)
                               VAR_DOS_SEQ.Device.PPJ203_PID.PID_Mode := FALSE;
                               VAR_DOS_SEQ.Device.PPJ203_PID.Auto_SP_Value := 0;
                               VAR_DOS_SEQ.Device.PPJ203_PID.FIX_Value := 0;

                               VAR_DOS_SEQ.Device.MMJ201_PID.PID_Enable := FALSE;                                      (* STEP: 153 Shaker Motor*)
                               VAR_DOS_SEQ.Device.MMJ201_PID.PID_Mode := FALSE;
                               VAR_DOS_SEQ.Device.MMJ201_PID.Auto_SP_Value := 0;
                               VAR_DOS_SEQ.Device.MMJ201_PID.FIX_Value := 0;

                               VAR_DOS_SEQ.Device.RVJ201_PID.PID_Enable := FALSE;                                      (* STEP: 153 *)
                               VAR_DOS_SEQ.Device.RVJ201_PID.PID_Mode := FALSE;
                               VAR_DOS_SEQ.Device.RVJ201_PID.Auto_SP_Value := 0;
                               VAR_DOS_SEQ.Device.RVJ201_PID.FIX_Value := 0;

                               VAR_DOS_SEQ.Device.AVJ201.AutoCnd := FALSE;                                             (* STEP: 153 Inlet Valve*)
                               VAR_DOS_SEQ.Device.AVJ201.EnableCnd := FALSE;
                               VAR_DOS_SEQ.Device.AVJ210.AutoCnd := FALSE;                                             (* STEP: 153 Washing Duct Valve*)
                               VAR_DOS_SEQ.Device.AVJ210.EnableCnd := FALSE;
                               VAR_DOS_SEQ.Device.AVJ211.AutoCnd := FALSE;                                             (* STEP: 153 Sprayball Valve*)
                               VAR_DOS_SEQ.Device.AVJ211.EnableCnd := FALSE;
                               VAR_DOS_SEQ.Device.AVJ212.AutoCnd := FALSE;                                             (* STEP: 153 *)
                               VAR_DOS_SEQ.Device.AVJ212.EnableCnd := FALSE;
                               VAR_DOS_SEQ.Device.AVJ215.AutoCnd := FALSE;                                             (* STEP: 153 Atmospheric drain valve*)
                               VAR_DOS_SEQ.Device.AVJ215.EnableCnd := FALSE;
                               VAR_DOS_SEQ.Device.AVJ216.AutoCnd := FALSE;                                             (* STEP: 153 Recirculation Valve*)
                               VAR_DOS_SEQ.Device.AVJ216.EnableCnd := FALSE;
                               VAR_DOS_SEQ.Device.AVJ217.AutoCnd := FALSE;                                             (* STEP: 153 Tank Hema Drain Valve*)
                               VAR_DOS_SEQ.Device.AVJ217.EnableCnd := FALSE;
                               VAR_DOS_SEQ.Device.AVJ218.AutoCnd := FALSE;                                             (* STEP: 153 Recirculation Valve*)
                               VAR_DOS_SEQ.Device.AVJ218.EnableCnd := FALSE;
                               VAR_DOS_SEQ.Device.AVJ221.AutoCnd := FALSE;                                             (* STEP: 153 Inlet Loop Valve*)
                               VAR_DOS_SEQ.Device.AVJ221.EnableCnd := FALSE;
                               VAR_DOS_SEQ.Device.AVJ230.AutoCnd := FALSE;                                             (* STEP: 153 *)
                               VAR_DOS_SEQ.Device.AVJ230.EnableCnd := FALSE;
                               VAR_DOS_SEQ.Device.AVJ231.AutoCnd := FALSE;                                             (* STEP: 153 *)
                               VAR_DOS_SEQ.Device.AVJ231.EnableCnd := FALSE;
                               VAR_DOS_SEQ.Device.AVJ232.AutoCnd := FALSE;                                             (* STEP: 153 *)
                               VAR_DOS_SEQ.Device.AVJ232.EnableCnd := FALSE;
                               VAR_DOS_SEQ.Device.AVJ233.AutoCnd := FALSE;                                             (* STEP: 153 *)
                               VAR_DOS_SEQ.Device.AVJ233.EnableCnd := FALSE;
                               VAR_DOS_SEQ.Device.AVJ234.AutoCnd := FALSE;                                             (* STEP: 153 *)
                               VAR_DOS_SEQ.Device.AVJ234.EnableCnd := FALSE;
                               VAR_DOS_SEQ.Device.AVJ235.AutoCnd := FALSE;                                             (* STEP: 153 *)
                               VAR_DOS_SEQ.Device.AVJ235.EnableCnd := FALSE;

                               VAR_DOS_SEQ.Device.LTJ203.ALR_HighLimitEn := FALSE;                                     (* STEP: 153 Hema Tank Level*)
                               VAR_DOS_SEQ.Device.LTJ203.ALR_HighLimitSP := 0;
                               VAR_DOS_SEQ.Device.LTJ203.ALR_LowLimitEn := FALSE;
                               VAR_DOS_SEQ.Device.LTJ203.ALR_LowLimitSP := 0;
                               VAR_DOS_SEQ.Device.LTJ203.SP := 0;
                               VAR_DOS_SEQ.Device.LTJ203.CMP := 0;
                               VAR_DOS_SEQ.Device.LTJ203.MinDev := 0;
                               VAR_DOS_SEQ.Device.LTJ203.MaxDev := 0;

                               VAR_DOS_SEQ.Device.TTJ203.ALR_HighLimitEn := FALSE;                                     (* STEP: 153 Hema Tank Temperature*)
                               VAR_DOS_SEQ.Device.TTJ203.ALR_HighLimitSP := 0;
                               VAR_DOS_SEQ.Device.TTJ203.ALR_LowLimitEn := FALSE;
                               VAR_DOS_SEQ.Device.TTJ203.ALR_LowLimitSP := 0;
                               VAR_DOS_SEQ.Device.TTJ203.SP := 0;
                               VAR_DOS_SEQ.Device.TTJ203.CMP := 0;
                               VAR_DOS_SEQ.Device.TTJ203.MinDev := 0;
                               VAR_DOS_SEQ.Device.TTJ203.MaxDev := 0;

                               VAR_DOS_SEQ.Device.LSJ200.ALR := FALSE;                                                 (* STEP: 153 *)
                               VAR_DOS_SEQ.Device.LSJ200.WAIT_OFF := FALSE;
                               VAR_DOS_SEQ.Device.LSJ200.WAIT_ON := FALSE;

                               VAR_DOS_SEQ.Device.LSJ201.ALR := FALSE;                                                 (* STEP: 153 *)
                               VAR_DOS_SEQ.Device.LSJ201.WAIT_OFF := FALSE;
                               VAR_DOS_SEQ.Device.LSJ201.WAIT_ON := FALSE;

                               VAR_DOS_SEQ.Device.LSJ202.ALR := FALSE;                                                 (* STEP: 153 *)
                               VAR_DOS_SEQ.Device.LSJ202.WAIT_OFF := FALSE;
                               VAR_DOS_SEQ.Device.LSJ202.WAIT_ON := FALSE;

                               VAR_DOS_SEQ.Device.FSJ201.ALR := FALSE;                                                 (* STEP: 153 *)
                               VAR_DOS_SEQ.Device.FSJ201.WAIT_OFF := FALSE;
                               VAR_DOS_SEQ.Device.FSJ201.WAIT_ON := FALSE;

                               VAR_DOS_SEQ.Device.FSJ202.ALR := FALSE;                                                 (* STEP: 153 *)
                               VAR_DOS_SEQ.Device.FSJ202.WAIT_OFF := FALSE;
                               VAR_DOS_SEQ.Device.FSJ202.WAIT_ON := FALSE;

                               VAR_DOS_SEQ.Mem.PBAbortEnable := FALSE;                                                 (* STEP: 153 PB Abort Sequence Enable*)
                               VAR_DOS_SEQ.Mem.PBStopEnable := TRUE;                                                   (* STEP: 153 PB Stop Sequence Enable*)
                               VAR_DOS_SEQ.Mem.PBStartEnable := FALSE;                                                 (* STEP: 153 PB Start Sequence Enable*)
                               VAR_DOS_SEQ.Mem.ContainersStop := FALSE;                                                (* STEP: 153 *)
                               VAR_DOS_SEQ.Mem.MachineStart := FALSE;                                                  (* STEP: 153 *)
                               VAR_DOS_SEQ.Mem.MachineStop := FALSE;                                                   (* STEP: 153 *)
                               VAR_DOS_SEQ.Mem.DummyBottles := FALSE;                                                  (* STEP: 153 Dummy Bottle Install*)
                               VAR_DOS_SEQ.Mem.PositioningRequest := FALSE;                                            (* STEP: 153 Request of Cam Positioning at height SP of Sequncer*)
                               VAR_DOS_SEQ.Mem.COP_Cycle := FALSE;                                                     (* STEP: 153 COP Cycle Check Requested*)
                               VAR_DOS_SEQ.Mem.LapsCounter := FALSE;                                                   (* STEP: 153 *)
                               VAR_DOS_SEQ.Mem.ValveOpening := FALSE;                                                  (* STEP: 153 *)
                               VAR_DOS_SEQ.Mem.CopAfterCipRequest := FALSE;                                            (* STEP: 153 Request Of Cop After Cip*)
```
